FUNCTION_BLOCK FB_ModbusManager_1

VAR
	fbModbusMaster: FB_ModbusMaster_R2;
	
	
	
	aRequests_Read: 			ARRAY[0..(GVL.Max_Modbus_Requests_Read - 1)] OF POINTER TO ST_Modbus_ReadRequest;
	nIterator_Read_Insert: 		INT := 0;
	nIterator_Read_Action: 		INT := 0;
	nTotalRequests_Read: 		INT := 0;
	
	aRequests_Write: 			ARRAY[0..(GVL.Max_Modbus_Requests_Write - 1)] OF POINTER TO ST_Modbus_WriteRequest;
	nIterator_Write_Insert: 	INT := 0;
	nIterator_Write_Action:		INT := 0;
	nTotalRequests_Write: 		INT := 0;
	
	nNumRetries: 				INT := 0;
	bRead_or_Write_0_1:			BOOL := FALSE;
	bRequestAccepted: 			BOOL := FALSE;
	
	eSMState: (WAIT, REQUEST_READ, READING, READ, REQUEST_WRITE, WRITING, WRITTEN, REQUEST_READ_PRIORITY, READING_PRIORITY, READ_PRIORITY, REQUEST_WRITE_PRIORITY, WRITING_PRIORITY, WRITTEN_PRIORITY,ERROR) := WAIT;
	
	fbTON_RequestTimeout: TON := (PT := GVL.ModbusTimeout);
	tDelayBetweenMsg:	TIME := T#100MS;	
	fbTON_DelayBetweenMSG: TON := (PT := tDelayBetweenMsg, IN := FALSE);
	
	
	// These two buffers are for priority messages and will be serviced before requests in the other buffers (similar to QoS)
	aRequests_Read_Priority: 			ARRAY[0..(GVL.Max_Modbus_Requests_Read_Priority - 1)] OF POINTER TO ST_Modbus_ReadRequest;
	nIterator_Read_Insert_Priority: 	INT := 0;
	nIterator_Read_Action_Priority: 	INT := 0;
	nTotalRequests_Read_Priority: 		INT := 0;
	
	aRequests_Write_Priority: 			ARRAY[0..(GVL.Max_Modbus_Requests_Write_Priority - 1)] OF POINTER TO ST_Modbus_WriteRequest;
	nIterator_Write_Insert_Priority: 	INT := 0;
	nIterator_Write_Action_Priority:	INT := 0;
	nTotalRequests_Write_Priority: 		INT := 0;
	
	bRead_or_Write_0_1_Priority:		BOOL := FALSE;
	
END_VAR

fbModbusMaster();
fbTON_RequestTimeout(PT := GVL.ModbusTimeout);


CASE eSMState OF
	
	WAIT:
		// Wait for a message to be received in either the Rx or Tx buffers
		nNumRetries := 0;
		fbTON_DelayBetweenMSG(PT := tDelayBetweenMsg, IN := TRUE);
		
		IF fbTON_DelayBetweenMSG.Q THEN
			// Service priority writes first
			IF nTotalRequests_Write_Priority > 0 THEN
				eSMState := REQUEST_WRITE_PRIORITY;
			// Service priority reads second
			ELSIF nTotalRequests_Read_Priority > 0 THEN
				eSMState := REQUEST_READ_PRIORITY;
			// Else toggle betwweenm read and write
			ELSIF bRead_or_Write_0_1 THEN   // If there are no priority messages then serve the non-critical requests
				bRead_or_Write_0_1 := FALSE;
				IF nTotalRequests_Write > 0 THEN
					eSMState := REQUEST_WRITE;
				END_IF
			ELSE 
				bRead_or_Write_0_1 := TRUE;
				IF nTotalRequests_Read > 0 THEN
					eSMState := REQUEST_READ;	
				END_IF
			END_IF
			fbTON_DelayBetweenMSG.IN := FALSE;
		END_IF
		

		
	REQUEST_READ:
		fbModbusMaster.readRegs(ReadRequest := aRequests_Read[nIterator_Read_Action], bRequestAccepted => bRequestAccepted);
		IF bRequestAccepted THEN
			eSMState := READING;
			bRequestAccepted := FALSE;
			fbTON_RequestTimeout.IN := TRUE;
		END_IF
		// Send a read request to the modbus master, progress to READING if modbus master accepts
		
	READING:
	
		IF aRequests_Read[nIterator_Read_Action]^.bRequestCompleted = TRUE THEN
			eSMState := READ;
			fbTON_RequestTimeout.IN := FALSE;
		END_IF
		
		IF fbTON_RequestTimeout.Q THEN
			eSMState := REQUEST_READ; 
			nNumRetries := nNumRetries + 1;
			IF nNumRetries > GVL.ModbusMaxRetires THEN
				// ADD CODE HERE - Raise an error - and proceed to the next request - attach info about the request to the error so we can troubleshoot it
				eSMState := READ;
			END_IF
		END_IF
		
		// Stay in this state until the boolean pointer of job completed is set to true
		// Monitor the timeout timer and retry request if necessary
		
	READ:
		// Set the position in the ring buffer to 0 and iterate to the next, return to wait where the decision will be made to read or write
		aRequests_Read[nIterator_Read_Action] := 0;
		nIterator_Read_Action := nIterator_Read_Action + 1;
		
		IF nIterator_Read_Action > (GVL.Max_Modbus_Requests_Read - 1) THEN // return to 0 index if we are at the end of the buffer
			nIterator_Read_Action := 0;
		END_IF
		nTotalRequests_Read := nTotalRequests_Read - 1;
		eSMState := WAIT;
	
		
	REQUEST_WRITE:
		// Send a read request to the modbus master, progress to WRITING if modbus master accepts
		fbModbusMaster.writeRegs(WriteRequest := aRequests_Write[nIterator_Write_Action], bRequestAccepted => bRequestAccepted);
		IF bRequestAccepted THEN
			eSMState := WRITING;
			bRequestAccepted := FALSE;
			fbTON_RequestTimeout.IN := TRUE;
		END_IF
		
	WRITING:
		// Stay in this state until the boolean pointer of job completed is set to true
		IF aRequests_Write[nIterator_Write_Action]^.bRequestCompleted = TRUE THEN
			eSMState := WRITTEN;
			fbTON_RequestTimeout.IN := FALSE;
		END_IF
		
		IF fbTON_RequestTimeout.Q THEN
			eSMState := REQUEST_WRITE; 
			nNumRetries := nNumRetries + 1;
			IF nNumRetries > GVL.ModbusMaxRetires THEN
				// ADD CODE HERE - Raise an error - and proceed to the next request - attach info about the request to the error so we can troubleshoot it
				eSMState := WRITTEN;
			END_IF
		END_IF
		
		
	WRITTEN:
		// Set the position in the ring buffer to 0 and iterate to the next, return to wait where the decision will be made to read or write
		aRequests_Write[nIterator_Write_Action] := 0;
		nIterator_Write_Action := nIterator_Write_Action + 1;
		
		IF nIterator_Write_Action > (GVL.Max_Modbus_Requests_Write - 1) THEN
			nIterator_Write_Action := 0;
		END_IF
		
		nTotalRequests_Write := nTotalRequests_Write - 1;
		eSMState := WAIT;
		
		
	REQUEST_READ_PRIORITY:
		fbModbusMaster.readRegs(ReadRequest := aRequests_Read_Priority[nIterator_Read_Action_Priority], bRequestAccepted => bRequestAccepted);
		IF bRequestAccepted THEN
			eSMState := READING_PRIORITY;
			bRequestAccepted := FALSE;
			fbTON_RequestTimeout.IN := TRUE;
		END_IF
		// Send a read request to the modbus master, progress to READING if modbus master accepts
		
	READING_PRIORITY:
	
		IF aRequests_Read_Priority[nIterator_Read_Action_Priority]^.bRequestCompleted = TRUE THEN
			eSMState := READ_PRIORITY;
			fbTON_RequestTimeout.IN := FALSE;
		END_IF
		
		IF fbTON_RequestTimeout.Q THEN
			eSMState := REQUEST_READ_PRIORITY; 
			nNumRetries := nNumRetries + 1;
			IF nNumRetries > GVL.ModbusMaxRetires THEN
				// ADD CODE HERE - Raise an error - and proceed to the next request - attach info about the request to the error so we can troubleshoot it
				eSMState := READ_PRIORITY;
			END_IF
		END_IF
		
		// Stay in this state until the boolean pointer of job completed is set to true
		// Monitor the timeout timer and retry request if necessary
		
	READ_PRIORITY:
		// Set the position in the ring buffer to 0 and iterate to the next, return to wait where the decision will be made to read or write
		aRequests_Read_Priority[nIterator_Read_Action_Priority] := 0;
		nIterator_Read_Action_Priority := nIterator_Read_Action_Priority + 1;
		
		IF nIterator_Read_Action_Priority > (GVL.Max_Modbus_Requests_Read_Priority - 1) THEN // return to 0 index if we are at the end of the buffer
			nIterator_Read_Action_Priority := 0;
		END_IF
		nTotalRequests_Read_Priority := nTotalRequests_Read_Priority - 1;
		eSMState := WAIT;
	
		
	REQUEST_WRITE_PRIORITY:
		// Send a read request to the modbus master, progress to WRITING if modbus master accepts
		fbModbusMaster.writeRegs(WriteRequest := aRequests_Write_Priority[nIterator_Write_Action_Priority], bRequestAccepted => bRequestAccepted);
		IF bRequestAccepted THEN
			eSMState := WRITING_PRIORITY;
			bRequestAccepted := FALSE;
			fbTON_RequestTimeout.IN := TRUE;
		END_IF
		
	WRITING_PRIORITY:
		// Stay in this state until the boolean pointer of job completed is set to true
		IF aRequests_Write_Priority[nIterator_Write_Action_Priority]^.bRequestCompleted = TRUE THEN
			eSMState := WRITTEN_PRIORITY;
			fbTON_RequestTimeout.IN := FALSE;
		END_IF
		
		IF fbTON_RequestTimeout.Q THEN
			eSMState := REQUEST_WRITE_PRIORITY; 
			nNumRetries := nNumRetries + 1;
			IF nNumRetries > GVL.ModbusMaxRetires THEN
				// ADD CODE HERE - Raise an error - and proceed to the next request - attach info about the request to the error so we can troubleshoot it
				eSMState := WRITTEN_PRIORITY;
			END_IF
		END_IF
		
		
	WRITTEN_PRIORITY:
		// Set the position in the ring buffer to 0 and iterate to the next, return to wait where the decision will be made to read or write
		aRequests_Write_Priority[nIterator_Write_Action_Priority] := 0;
		nIterator_Write_Action_Priority := nIterator_Write_Action_Priority + 1;
		
		IF nIterator_Write_Action_Priority > (GVL.Max_Modbus_Requests_Write_Priority - 1) THEN
			nIterator_Write_Action_Priority := 0;
		END_IF
		
		nTotalRequests_Write_Priority := nTotalRequests_Write_Priority - 1;
		eSMState := WAIT;
		
	ERROR:
		//
		
END_CASE

METHOD addRequest_Read : BOOL
VAR_INPUT
	ReadRequest: POINTER TO ST_Modbus_ReadRequest;
END_VAR
IF aRequests_Read[nIterator_Read_Insert] = 0 THEN
	
	aRequests_Read[nIterator_Read_Insert] := ReadRequest;
	aRequests_Read[nIterator_Read_Insert]^.bRequestAccepted := FALSE;
	aRequests_Read[nIterator_Read_Insert]^.bRequestCompleted := FALSE;
	nIterator_Read_Insert := nIterator_Read_Insert + 1;
	
	IF nIterator_Read_Insert > (GVL.Max_Modbus_Requests_Read -1) THEN
		nIterator_Read_Insert := 0;
	END_IF
	
	nTotalRequests_Read := nTotalRequests_Read + 1;
	
	
	addRequest_Read := TRUE;
ELSE
	addRequest_Read := FALSE;	// A buffer overflow has occured here, add some error raising code here
END_IF
END_METHOD

METHOD addRequest_Read_Priority : BOOL
VAR_INPUT
	ReadRequest: POINTER TO ST_Modbus_ReadRequest;
END_VAR
IF aRequests_Read_Priority[nIterator_Read_Insert_Priority] = 0 THEN
	
	aRequests_Read_Priority[nIterator_Read_Insert_Priority] := ReadRequest;
	aRequests_Read_Priority[nIterator_Read_Insert_Priority]^.bRequestAccepted := FALSE;
	aRequests_Read_Priority[nIterator_Read_Insert_Priority]^.bRequestCompleted := FALSE;
	nIterator_Read_Insert_Priority := nIterator_Read_Insert_Priority + 1;
	
	IF nIterator_Read_Insert_Priority > (GVL.Max_Modbus_Requests_Read_Priority -1) THEN
		nIterator_Read_Insert_Priority := 0;
	END_IF
	
	nTotalRequests_Read_Priority := nTotalRequests_Read_Priority + 1;
	
	
	addRequest_Read_Priority := TRUE;
ELSE
	addRequest_Read_Priority := FALSE;	// A buffer overflow has occured here, add some error raising code here
END_IF
END_METHOD

METHOD addRequest_Write : BOOL
VAR_INPUT
	WriteRequest: POINTER TO ST_Modbus_WriteRequest;
END_VAR
IF aRequests_Write[nIterator_Write_Action] = 0 THEN
	aRequests_Write[nIterator_Write_Action] := WriteRequest;
	aRequests_Write[nIterator_Write_Action]^.bRequestAccepted := FALSE;
	aRequests_Write[nIterator_Write_Action]^.bRequestCompleted := FALSE;
	nIterator_Write_Insert := nIterator_Write_Insert + 1;
	
	IF nIterator_Write_Insert > (GVL.Max_Modbus_Requests_Write - 1) THEN
		nIterator_Write_Insert := 0;
	END_IF
	
	nTotalRequests_Write := nTotalRequests_Write + 1;
	
ELSE
	addRequest_Write := FALSE; // A buffer overflow has occured here, add some error raising code here
END_IF
END_METHOD

METHOD addRequest_Write_Priority : BOOL
VAR_INPUT
	WriteRequest: POINTER TO ST_Modbus_WriteRequest;
END_VAR
IF aRequests_Write_Priority[nIterator_Write_Insert_Priority] = 0 THEN
	
	aRequests_Write_Priority[nIterator_Write_Insert_Priority] := WriteRequest;
	aRequests_Write_Priority[nIterator_Write_Insert_Priority]^.bRequestAccepted := FALSE;
	aRequests_Write_Priority[nIterator_Write_Insert_Priority]^.bRequestCompleted := FALSE;
	nIterator_Write_Insert_Priority := nIterator_Write_Insert_Priority + 1;
	
	IF nIterator_Write_Insert_Priority > (GVL.Max_Modbus_Requests_Write_Priority - 1) THEN
		nIterator_Write_Insert_Priority := 0;
	END_IF
	
	nTotalRequests_Write_Priority := nTotalRequests_Write_Priority + 1;
	
ELSE
	addRequest_Write_Priority := FALSE; // A buffer overflow has occured here, add some error raising code here
END_IF
END_METHOD

METHOD FB_init : BOOL
VAR_INPUT
	bInitRetains : BOOL; // if TRUE, the retain variables are initialized (warm start / cold start)
	bInCopyCode : BOOL;  // if TRUE, the instance afterwards gets moved into the copy code (online change)
END_VAR

VAR
	i: INT := 0;
END_VAR
WHILE i < GVL.Max_Modbus_Requests_Read DO
	aRequests_Read[i] := 0;
	i := i + 1;
END_WHILE

i := 0;

WHILE i < GVL.Max_Modbus_Requests_Write DO
	aRequests_Write[i] := 0;
	i := i + 1;
END_WHILE
END_METHOD

END_FUNCTION_BLOCK

(* stored: Version 1.1.0.1, ProductVersion 3.1.4024.12
   POU FB_ModbusManager_1: Id {a45a9f6f-9eeb-450c-8aef-ce77e8229394}, SpecialFunc None
   Method addRequest_Read: Id {ad48a1a4-52f1-4dea-8eef-87901e557945}
   Method addRequest_Read_Priority: Id {5d20d996-824d-49c7-89b2-c2693d62c621}
   Method addRequest_Write: Id {3e3e0419-59c7-4e12-9c84-5505a6f189ea}
   Method addRequest_Write_Priority: Id {93705f01-623c-42d3-a2af-300eac560b80}
   Method FB_init: Id {56d5ca7a-5c7b-4e63-b956-3bdc9d4f668b} *)
